//{attribute 'qualified_only'}
{attribute 'strict'}
{attribute 'to_string'}
TYPE E_State :
(
	IDLE,
	STARTING,
	EXECUTE,
	HOLDING,
	UNHOLDING,
	HELD,
	COMPLETING,
	COMPLETED,
	RESETTING,
	ABORTING,
	ABORTED,
	CLEARING,
	STOPPING,
	STOPPED	
);
END_TYPE

(* stored: Version 1.1.0.1
   DUT E_State: Id {b1c5ce1b-cacd-4233-aae4-fe81a7be0f16} *)
